REGION Network 4: Block description — Section 3.5 to 3.5
   // ▂▂▂▂▂▂▂▂▂▂▂▂▂▂▂▂▂▂▂▂▂▂▂▂▂▂▂▂▂▂▂▂▂▂▂▂▂▂▂▂▂▂▂▂
   // 3.5     Expressing the calculations in Controller operations
   // 
   // The calculations above must be rendered in a form suitable for the Simatic S7-1500 Controller, 
   // using the mathematical operations available to that Controller, these are listed in Table 2.1.
   // 
   // To perform the calculations in the Controller it will be necessary to use partial calculation to 
   // hold separate components of the overall calculation and combine these to produce the final 
   // result. 
   // 
   // The following sections breakdown each of the response calculations into these partial 
   // calculations and demonstrate how these are then combined to provide a final result that is 
   // compatible with the Controller mathematical operations and Controller notations.
   // 
   // 
   // 
   // ▁▁▁▁▁▁▁▁▁▁▁▁▁▁▁▁▁▁▁▁▁▁▁▁▁▁▁▁▁▁▁▁▁▁▁▁▁▁▁▁▁▁▁▁
   // 3.5.1     Over damped, slow response no overshoot             ζ > 1
   // 
   // 
   // CALCULATION:
   // 
   //       ╓   1 ┌   ζ       ┐   - ω [ ζ ─ √(ζ² ─ 1) ]t       1 ┌   ζ       ┐   - ω [ ζ ┼ √(ζ² ─ 1) ]t ╖
   // y(t) = K║x(t) ─ -- │------------------ ┼ 1│ｅ         ┼ -- │------------------ ─ 1│ｅ           ║
   //       ╙   2 └ √(ζ² ─ 1)     ┘            2 └ √(ζ² ─ 1)     ┘            ╜
   // 
   // 
   // 
   // Is rendered into the correct format as follows:
   // 
   // 
   //  cal_01 = SQRT ( SQR (ζ) - 1)         = √(ζ² ─ 1)
   // 
   //                                  ζ
   //  cal_02 = ζ ÷ cal_01              = -----------------
   //                          √(ζ² ─ 1)
   // 
   //  cal_03 = ζ + cal_01              = ζ ┼ √(ζ² ─ 1)
   // 
   //  cal_04 = -1 × ω × t × cal_03           = - ω [ ζ ┼ √(ζ² ─ 1) ]t
   // 
   //                              -ω [ ζ ┼ √(ζ² ─ 1) ]t 
   //  cal_05 = EXP( cal_04 )              =ｅ
   // 
   //  cal_06 = ζ - cal_01               = ζ ─ √(ζ² ─ 1)
   // 
   //  cal_07 = -1 × ω × t × cal_06           = - ω [ ζ ─ √(ζ² ─ 1) ]t
   // 
   //                            -ω [ ζ ─ √(ζ² ─ 1) ]t 
   //  cal_08 = EXP( cal_07 )              =ｅ
   // 
   //                           1 ┌   ζ       ┐
   //  cal_09 = (cal_02 - 1) × 0.5           = -- │------------------ ─ 1│
   //                           2 └ √(ζ² ─ 1)     ┘
   // 
   //                           1 ┌   ζ       ┐
   //  cal_10 = (cal_02 + 1) × 0.5            = -- │------------------ ┼ 1│
   //                           2 └ √(ζ² ─ 1)     ┘
   // 
   //                           1 ┌   ζ       ┐   -ω [ ζ ┼ √(ζ² ─ 1) ]t
   //  cal_11 = cal_09 × cal_05             = -- │------------------ ─ 1│ｅ
   //                           2 └ √(ζ² ─ 1)     ┘
   // 
   //                           1 ┌   ζ       ┐   -ω [ ζ ─ √(ζ² ─ 1) ]t
   //  cal_12 = cal_10 × cal_08             = -- │------------------ ┼ 1│ｅ
   //                           2 └ √(ζ² ─ 1)     ┘
   // 
   //                          ╓   1 ┌   ζ       ┐   - ω [ ζ ─ √(ζ² ─ 1) ]t       1 ┌   ζ       ┐   - ω [ ζ ┼ √(ζ² ─ 1) ]t ╖
   //  cal_13 = INPUT - cal_12 + cal_11        = ║x(t) ─ -- │------------------ ┼ 1│ｅ         ┼ -- │------------------ ─ 1│ｅ           ║
   //                          ╙   2 └ √(ζ² ─ 1)     ┘            2 └ √(ζ² ─ 1)     ┘            ╜
   // 
   //                             ╓   1 ┌   ζ       ┐   - ω [ ζ ─ √(ζ² ─ 1) ]t       1 ┌   ζ       ┐   - ω [ ζ ┼ √(ζ² ─ 1) ]t ╖
   //  OUTPUT  = K × cal_13             =  K║x(t) ─ -- │------------------ ┼ 1│ｅ         ┼ -- │------------------ ─ 1│ｅ           ║
   //                             ╙   2 └ √(ζ² ─ 1)     ┘            2 └ √(ζ² ─ 1)     ┘            ╜
   // 
   // 
   // 
   // ▁▁▁▁▁▁▁▁▁▁▁▁▁▁▁▁▁▁▁▁▁▁▁▁▁▁▁▁▁▁▁▁▁▁▁▁▁▁▁▁▁▁▁▁
   // 3.5.2     Critically damped, fastest response without overshoot        ζ = 1
   // 
   // 
   // CALCULATION:
   // 
   //       ╓           - ωt  ╖
   // y(t) = K║x(t) ─ (1 ┼ ωt) ｅ  ║
   //       ╙             ╜
   // 
   // 
   // Is rendered into the correct format as follows:
   // 
   // 
   //  cal_01 = -1 × ω × t                = - ωt  
   // 
   //                          - ωt
   //  cal_02 = EXP( cal_01 )              =ｅ
   // 
   //  cal_03 = 1 - cal_01              = 1 ─ (-ωt) = 1 ┼ ωt
   // 
   //                              - ωt
   //  cal_04 = cal_03 × cal_02            = (1 ┼ ωt) ｅ
   // 
   //                                 - ωt
   //  cal_05 = INPUT  - cal_04            = x(t) ─ (1 ┼ ωt) ｅ
   // 
   //                             ╓           - ωt  ╖
   //  OUTPUT  = K × cal_05             =  K║x(t) ─ (1 ┼ ωt) ｅ  ║
   //                             ╙             ╜
   // 
   // 
   // 
   // ▁▁▁▁▁▁▁▁▁▁▁▁▁▁▁▁▁▁▁▁▁▁▁▁▁▁▁▁▁▁▁▁▁▁▁▁▁▁▁▁▁▁▁▁
   // 3.5.3     Under damped, decreasing oscillations              0 < ζ < 1
   // 
   // 
   // CALCULATION:
   // 
   //       ╓      - ζω t  ┌        ζ            ┐╖
   // y(t) = K║x(t) ─ ｅ   │COS (Ωt) ┼ ------------------ SIN (Ωt)│║  where Ω =  ω √(1 ─ ζ²)
   //       ╙       └       √(1 ─ ζ²)       ┘╜
   // 
   // 
   // Is rendered into the correct format as follows:
   // 
   // 
   //  cal_01 = SQRT ( 1 - SQR (ζ))         = √(1 ─ ζ²)
   // 
   //                                  ζ
   //  cal_02 = ζ ÷ cal_01              = -----------------
   //                          √(1 ─ ζ²)
   // 
   //  cal_03 = ω × cal_01                = ω √(1 ─ ζ²) = Ω
   // 
   //  cal_04 = t × cal_03              = Ωt
   // 
   //  cal_05 = COS( cal_04 )             = COS (Ωt)
   // 
   //  cal_06 = SIN( cal_04 )               = SIN (Ωt)
   // 
   //  cal_07 = -1 × ζ × ω × t             = - ζω t 
   // 
   //                          - ζω t 
   //  cal_08 = EXP( cal_07 )              =ｅ
   // 
   //                          - ζω t 
   //  cal_09 = cal_08 × cal_05            =ｅ         COS (Ωt)
   // 
   //  
   //                                  ζ      - ζω t
   //  cal_10 = cal_02 × cal_08 × cal_06        = ----------------- ｅ         SIN (Ωt)
   //                          √(1 ─ ζ²)
   // 
   //                            ╓      - ζω t          ζ     - ζω t            ╖  ╓      - ζω t  ┌        ζ            ┐╖
   //  cal_11 = INPUT - cal_09 - cal_10          =║x(t) ─ ｅ   COS (Ωt) ─ ------------------ ｅ   SIN (Ωt)║=║x(t) ─ ｅ   │COS (Ωt) ┼ ------------------ SIN (Ωt)│║
   //                            ╙              √(1 ─ ζ²)              ╜  ╙       └       √(1 ─ ζ²)       ┘╜
   // 
   //                             ╓      - ζω t  ┌        ζ            ┐╖
   //  OUTPUT  = K × cal_11             =  K║x(t) ─ ｅ   │COS (Ωt) ┼ ------------------ SIN (Ωt)│║
   //                             ╙       └       √(1 ─ ζ²)       ┘╜
   // 
   // 
   // 
   // ▁▁▁▁▁▁▁▁▁▁▁▁▁▁▁▁▁▁▁▁▁▁▁▁▁▁▁▁▁▁▁▁▁▁▁▁▁▁▁▁▁▁▁▁
   // 3.5.4     Undamped, oscillates with frequency ω              ζ = 0
   // 
   // 
   // CALCULATION:
   // 
   //       ╓       ╖
   // y(t) = K║x(t) ─ COS (ωt) ║
   //       ╙       ╜
   // 
   // 
   // Is rendered into the correct format as follows:
   // 
   // 
   //  cal_01 = ω × t                  = ωt
   // 
   //  cal_02 = COS( cal_01 )             = COS (ωt)
   // 
   //  cal_03 = INPUT - cal_02             = x(t) ─ COS (ωt) 
   // 
   //  OUTPUT  = K × cal_03             =  K [ x(t) ─ COS (ωt) ]
   // 
   // 
   // 
   // ▁▁▁▁▁▁▁▁▁▁▁▁▁▁▁▁▁▁▁▁▁▁▁▁▁▁▁▁▁▁▁▁▁▁▁▁▁▁▁▁▁▁▁▁
   // 3.5.5     Unstable, oscillations of increasing amplitude           -1 < ζ < 0
   // 
   // 
   // CALCULATION:
   // 
   //       ╓      | ζ | ω t ┌        ζ            ┐╖
   // y(t) = K║x(t) ─ ｅ    │COS (Ωt) ┼ ------------------ SIN (Ωt)│║  where Ω =  ω √(1 ─ ζ²)
   //       ╙          └       √(1 ─ ζ²)       ┘╜
   // 
   // 
   // Is rendered into the correct format as follows:
   // 
   // 
   //  cal_01 = SQRT ( 1 - SQR (ζ))         = √(1 ─ ζ²)
   // 
   //                                  ζ
   //  cal_02 = ζ ÷ cal_01              = -----------------
   //                          √(1 ─ ζ²)
   // 
   //  cal_03 = ω × cal_01                = ω √(1 ─ ζ²) = Ω
   // 
   //  cal_04 = t × cal_03              = Ωt
   // 
   //  cal_05 = COS( cal_04 )             = COS (Ωt)
   // 
   //  cal_06 = SIN( cal_04 )               = SIN (Ωt)
   // 
   //  cal_07 = ABS(ζ) × ω × t              =  | ζ | ω t 
   // 
   //                           | ζ | ω t 
   //  cal_08 = EXP( cal_07 )              =ｅ
   // 
   //                           | ζ | ω t 
   //  cal_09 = cal_08 × cal_05            =ｅ         COS (Ωt)
   // 
   //  
   //                                  ζ      | ζ | ω t
   //  cal_10 = cal_02 × cal_08 × cal_06        = ----------------- ｅ         SIN (Ωt)
   //                          √(1 ─ ζ²)
   // 
   //                            ╓       | ζ | ω t         ζ      | ζ | ω t         ╖  ╓      | ζ | ω t ┌        ζ            ┐╖
   //  cal_11 = INPUT - cal_09 - cal_10          =║x(t) ─ ｅ   COS (Ωt) ─ ------------------ ｅ   SIN (Ωt)║=║x(t) ─ ｅ    │COS (Ωt) ┼ ------------------ SIN (Ωt)│║
   //                            ╙              √(1 ─ ζ²)              ╜  ╙        └       √(1 ─ ζ²)       ┘╜
   // 
   //                             ╓      | ζ | ω t ┌        ζ            ┐╖
   //  OUTPUT  = K × cal_11             =  K║x(t) ─ ｅ    │COS (Ωt) ┼ ------------------ SIN (Ωt)│║
   //                             ╙          └       √(1 ─ ζ²)       ┘╜
   // 
   // 
   // 
   // ▁▁▁▁▁▁▁▁▁▁▁▁▁▁▁▁▁▁▁▁▁▁▁▁▁▁▁▁▁▁▁▁▁▁▁▁▁▁▁▁▁▁▁▁
   // 3.5.6     Unstable, unbounded asymptotic increase              ζ ≤ -1
   // 
   // 
   // CALCULATION:
   // 
   //       ╓   1 ┌   ζ       ┐     ω [ | ζ | ─ √(ζ² ─ 1) ]t    1 ┌   ζ       ┐     ω [ | ζ | ┼ √(ζ² ─ 1) ]t ╖
   // y(t) = K║x(t) ─ -- │------------------ ┼ 1│ｅ         ┼ -- │------------------ ┼ 1│ｅ              ║
   //       ╙   2 └ √(ζ² ─ 1)     ┘            2 └ √(ζ² ─ 1)     ┘               ╜
   // 
   // 
   // 
   // Is rendered into the correct format as follows:
   // 
   // 
   //  cal_01 = SQRT ( SQR (ζ) - 1)         = √(ζ² ─ 1)
   // 
   //                                  ζ
   //  cal_02 = ζ ÷ cal_01              = -----------------
   //                          √(ζ² ─ 1)
   // 
   //  cal_03 = ABS (ζ) + cal_01            = | ζ | ┼ √(ζ² ─ 1)
   // 
   //  cal_04 = ω × t × cal_03             = ω [ | ζ | ┼ √(ζ² ─ 1) ]t
   // 
   //                               ω [ | ζ | ┼ √(ζ² ─ 1) ]t 
   //  cal_05 = EXP( cal_04 )              =ｅ
   // 
   //  cal_06 = ABS (ζ) - cal_01             =  | ζ | ─ √(ζ² ─ 1)
   // 
   //  cal_07 = ω × t × cal_06             = ω [  | ζ | ─ √(ζ² ─ 1) ]t
   // 
   //                               ω [  | ζ | ─ √(ζ² ─ 1) ]t 
   //  cal_08 = EXP( cal_07 )              =ｅ
   // 
   //                           1 ┌   ζ       ┐
   //  cal_09 = (cal_02 + 1) × 0.5            = -- │------------------ ┼ 1│
   //                           2 └ √(ζ² ─ 1)     ┘
   // 
   //                           1 ┌   ζ       ┐   -ω [ ζ ─ √(ζ² ─ 1) ]t
   //  cal_10 = cal_09 × cal_08             = -- │------------------ ┼ 1│ｅ
   //                           2 └ √(ζ² ─ 1)     ┘
   // 
   //                           1 ┌   ζ       ┐   -ω [ ζ ┼ √(ζ² ─ 1) ]t
   //  cal_11 = cal_09 × cal_05             = -- │------------------ ┼ 1│ｅ
   //                           2 └ √(ζ² ─ 1)     ┘
   // 
   //                          ╓   1 ┌   ζ       ┐   - ω [ ζ ─ √(ζ² ─ 1) ]t       1 ┌   ζ       ┐   - ω [ ζ ┼ √(ζ² ─ 1) ]t ╖
   //  cal_12 = INPUT - cal_10 + cal_11        = ║x(t) ─ -- │------------------ ┼ 1│ｅ         ┼ -- │------------------ ┼ 1│ｅ           ║
   //                          ╙   2 └ √(ζ² ─ 1)     ┘            2 └ √(ζ² ─ 1)     ┘            ╜
   // 
   //                             ╓   1 ┌   ζ       ┐   - ω [ ζ ─ √(ζ² ─ 1) ]t       1 ┌   ζ       ┐   - ω [ ζ ┼ √(ζ² ─ 1) ]t ╖
   //  OUTPUT  = K × cal_12             =  K║x(t) ─ -- │------------------ ┼ 1│ｅ         ┼ -- │------------------ ┼ 1│ｅ           ║
   //                             ╙   2 └ √(ζ² ─ 1)     ┘            2 └ √(ζ² ─ 1)     ┘            ╜
   // 
   // 
   // 
   // ▂▂▂▂▂▂▂▂▂▂▂▂▂▂▂▂▂▂▂▂▂▂▂▂▂▂▂▂▂▂▂▂▂▂▂▂▂▂▂▂▂▂▂▂
   // 3.6     Operating modes
   // 
   // 
   // This block FC19152_StdDebugInst2Order supports manual and automatic operating modes, the 
   // default mode is automatic.
   // 
   // The module can be switched between automatic and manual modes with the 
   // mode_AutMan signal:
   // 
   //  DATA STRUCTURE    UT39152_Dy_DebugInst2Order
   //  ――――――――――――――――――――――――――――――――――――――――――
   //  SIGNAL         FUNCTION               TYPE     DETAILS
   //  ――――――――――――――――――――――――――――――――――――――――――
   //  Mode_AutMan     Specifies the operating mode of     Bool  1 = automatic mode
   //            the simulation                 0 = manual mode
   // 
   //  Mode_Time       Specifies the manual time value of       Real     Elapsed time
   //            the simulation in seconds           in seconds
   // 
   //  status_Aut      The simulation is in automatic mode   Bool  1 = auto mode
   //                                  0 = no in auto
   // 
   //  status_Man       The simulation is in manual mode    Bool  1 = manual mode
   //                                  0 = no in manual
   //  ――――――――――――――――――――――――――――――――――――――――――  
   // 
   // 
   // 
   // ▁▁▁▁▁▁▁▁▁▁▁▁▁▁▁▁▁▁▁▁▁▁▁▁▁▁▁▁▁▁▁▁▁▁▁▁▁▁▁▁▁▁▁▁
   // 3.6.1    Automatic mode
   // 
   // 
   // By default the module will be in automatic mode. 
   // 
   // In automatic mode, if the simulation is active (TRIGGER = 1), the module carries out the relevant 
   // calculation (listed in § 3.2) depending on the value of the damping factor (k_DampFactor) each 
   // time the module is called. The module calculates the elapsed time based on the current CPU 
   // time when the module was called, compared with the CPU time when the simulation was 
   // started (rising edge of TRIGGER) and stored in actual_StartTime.
   // 
   // In automatic mode, a real time simulation occurs, generating responses similar to those shown 
   // in the plots of § 2.3.  
   // 
   // 
   // 
   // ▁▁▁▁▁▁▁▁▁▁▁▁▁▁▁▁▁▁▁▁▁▁▁▁▁▁▁▁▁▁▁▁▁▁▁▁▁▁▁▁▁▁▁▁
   // 3.6.2    Manual mode
   // 
   // 
   // In manual mode, if the simulation is active (TRIGGER = 1), the module carries out the relevant 
   // calculation (listed in § 3.2) depending on the value of the damping factor (k_DampFactor) each 
   // time the module is called; in exactly the same way as automatic mode.
   // 
   // The difference with manual mode, is that the time used in the calculation must be uniquely 
   // specified, the elapsed time is not calculated and a manual time value must be provided.
   // 
   // The manual time is given in the variable mode_ManTime and is specified in seconds.
   // 
   // If mode mode_ManTime remains constant between module calls, the module will return the 
   // same OUTPUT value each time (assuming all other signals remain unchanged).
   // 
   // Manual mode allows the module to calculate the correct response for a particular and exact time, 
   // and is not dependent on cycle times or other factors that may affect when the module is called.
   // 
   // 
   // 
   // ▁▁▁▁▁▁▁▁▁▁▁▁▁▁▁▁▁▁▁▁▁▁▁▁▁▁▁▁▁▁▁▁▁▁▁▁▁▁▁▁▁▁▁▁
   // 3.7      Symbols, block icons and faceplates
   // 
   // There is no supervisory system interface for this block. It is a debug simulation module and as
   // such has no  graphical symbol, block icon or faceplate.
   // 
   //                ━━━   ⬙⬙⬙⬙⬙⬙   ━━━
END_REGION

REGION Network 5: Block description — Sections 4 to 11
   // ▄▄▄▄▄▄▄▄▄▄▄▄▄▄▄▄▄▄▄▄▄▄▄▄▄▄▄▄▄▄▄▄▄▄▄▄▄▄▄▄▄▄▄▄
   // 4.     PARAMETERS
   // 
   // 
   // The following parameters are associated with the block:
   // 
   //  
   //  ――――――――――――――――――――――――――――――――――――――――――
   //  PARAM         FUNCTION                    TYPE      IN-OUT 
   //  ――――――――――――――――――――――――――――――――――――――――――
   //  SYS_SIGNALS      Common system signals              UT21000    In
   //           logic and timing signals for parametric access
   // 
   //  TRIGGER       Activates the simulation (the simulation will run     Bool      In
   //           whilever this signal is high), the elapsed time 
   //           is measured from the rising edge of this signal
   // 
   //  INPUT        The input time function, x(t) in the calculations     Real      In
   // 
   //  DYNAMIC_DATA      Data structure that holds the live data for the       UT39152    InOut
   //           simulation (damping factor, natural frequency, 
   //           system gain, elapsed time &c.)
   // 
   //  OUTPUT       The output time response, y(t) in the calculations   Real      Out
   //  ――――――――――――――――――――――――――――――――――――――――――
   // 
   //                ━━━   ⬙⬙⬙⬙⬙⬙   ━━━
   // 
   // 
   // 
   // ▄▄▄▄▄▄▄▄▄▄▄▄▄▄▄▄▄▄▄▄▄▄▄▄▄▄▄▄▄▄▄▄▄▄▄▄▄▄▄▄▄▄▄▄
   // 5.     DATA STRUCTURES AND USAGE (AND INSTANCE DATA BLOCKS)
   // 
   // 
   // The block has the following associated data structure:
   // 
   // 
   //  ――――――――――――――――――――――――――――――――――――――――――
   //  DATA STRUCTURE             DESCRIPTION
   //  ――――――――――――――――――――――――――――――――――――――――――
   //  UT01000_St_SysRevision          Revision information for this block    See FC01001
   //  UT01001_St_SysLicence           Licence information for this block  See FC01001
   //  UT21000_Dy_SysSignals           System signals for logic and timing  See FC01001
   // 
   //  UT39152_Dy_DebugInst2Orderl       Dynamic data storage, contains live data, such as 
   //                     calculation variables, elapsed time, oscillation 
   //                     frequency and status signals
   //  ――――――――――――――――――――――――――――――――――――――――――
   // 
   // 
   // ▂▂▂▂▂▂▂▂▂▂▂▂▂▂▂▂▂▂▂▂▂▂▂▂▂▂▂▂▂▂▂▂▂▂▂▂▂▂▂▂▂▂▂▂
   // 5.2      UT39152_Dy_DebugInst2Order
   // 
   // The static data structure for an isolating valve.
   // 
   // 
   // 
   //  UT39152_Dy_DebugInst2Order (full contents)
   //  ――――――――――――――――――――――――――――――――――――――――――
   //  SIGNAL NAME          FUNCTION                     TYPE
   //  ――――――――――――――――――――――――――――――――――――――――――
   //  k_Gain             CONSTANT — Simulation system gain        Real
   //  k_NatFreq          CONSTANT — Simulation natural frequency (rad/s)   Real
   //  k_DampFactor        CONSTANT — Simulation damping factor        Real
   //  status_Running      STATUS — Simulation is running  Bool
   //                      (1 = running, 0 = stopped)
   //  status_Stopped        STATUS — Simulation is stopped (not running)    Bool
   //                      (1 = stopped, 0 = running)
   //  status_Stable         STATUS — Simulation response type is stable     Bool
   //                      (1 = stable, 0 = unstable)
   //  status_OverDamp       STATUS — Response is stable/over damped      Bool
   //                      (1 = stable, over damped)
   //  status_CritDamp       STATUS — Response is stable/critically damped     Bool
   //                      (1 = stable, critically damped)
   //  status_UnderDamp     STATUS — Response is stable/under damped      Bool
   //                      (1 = stable, under damped)
   //  status_Undamped      STATUS — Response is stable/undamped       Bool
   //                      (1 = stable, undamped)
   //  status_USUnder        STATUS — Response is unstable/under damped    Bool
   //                      (1 = unstable, under damped)
   //  status_USOver       STATUS — Response is unstable/over damped    Bool
   //                      (1 = unstable, over damped)
   //  status_Osc          STATUS — Oscillatory response             Real
   //                      (1 = osc. response, 0 = non-osc.)
   //  status_OscFreqRS       STATUS — Frequency of oscillation, zero if       Real
   //                      non-oscillatory (rad/s)
   //  status_OscFreqHz       STATUS — Frequency of oscillation, zero if       Real
   //                      non-oscillatory (Hz)
   //  status_Period         STATUS — Period of oscillation, zero if           Real
   //                      non-oscillatory (s)
   //  status_Aut           STATUS — Simulation is in automatic mode      Bool
   //                      (1 = automatic, 0 = manual)
   //  status_Man          STATUS — Simulation is in manual mode        Bool
   //                      (1 = manual, 0 = automatic)
   //  cal_PeakValue          CALC — Peak output value             Real
   //  cal_NatPeriod        CALC — Period of natural oscillations (s)       Real
   //                    zero for non-oscillatory response
   //  cal_DampFreq       CALC — Damped frequency of the system (rad/s)    Real
   //  cal_DampFreqHz         CALC — Damped frequency of the system (Hz)     Real
   //  cal_DampPeriod       CALC — Period of damped oscillations (s)       Real
   //                    zero for non-oscillatory response
   //  cal_TimeSteady        CALC — Time to reach steady state (s)       Real
   //                    zero for unstable response
   //  cal_Time63%          CALC — Time to reach 63% of steady state (s)      Real
   //                    zero for unstable response
   //  cal_TimePeak            CALC — Time to reach the peak ouptut value (s)    Real
   //  mode_AutMan       MODE — Automatic/manual mode selection     Bool
   //                      (1 = auto mode, 0 = manual mode)
   //  mode_ManTime       MODE — Manual mode time value (s)        Real
   //  actual_StartTime         ACTUAL — CPU time when simulation started       Real
   //  actual_RunTime        ACTUAL — Elapsed time since the            Real
   //                      simulation started (s)
   //  ――――――――――――――――――――――――――――――――――――――――――
   // 
   // 
   //                ━━━   ⬙⬙⬙⬙⬙⬙   ━━━
   // 
   // 
   // 
   // ▄▄▄▄▄▄▄▄▄▄▄▄▄▄▄▄▄▄▄▄▄▄▄▄▄▄▄▄▄▄▄▄▄▄▄▄▄▄▄▄▄▄▄▄
   // 6.     CONSTANTS AND TEMPORARY (LOCAL) DATA
   // 
   // There is no constant data.
   // 
   // The following temporary data is used:
   // 
   //  Temporary (local) data
   //  ――――――――――――――――――――――――――――――――――――――――――
   //  SIGNAL NAME          FUNCTION                  TYPE
   //  ――――――――――――――――――――――――――――――――――――――――――
   //  revInfo             Revision information for the block         UT01000
   //  licInfo           Licensing information for the block      UT01001
   //  cal_01          Partial calculation see § 3.5 for details      Real
   //  cal_02          Partial calculation see § 3.5 for details      Real
   //  cal_03          Partial calculation see § 3.5 for details      Real
   //  cal_04          Partial calculation see § 3.5 for details      Real
   //  cal_05          Partial calculation see § 3.5 for details      Real
   //  cal_06          Partial calculation see § 3.5 for details      Real
   //  cal_07          Partial calculation see § 3.5 for details      Real
   //  cal_08          Partial calculation see § 3.5 for details      Real
   //  cal_09          Partial calculation see § 3.5 for details      Real
   //  cal_10          Partial calculation see § 3.5 for details      Real
   //  cal_11          Partial calculation see § 3.5 for details      Real
   //  cal_12          Partial calculation see § 3.5 for details      Real
   //  cal_13          Partial calculation see § 3.5 for details      Real
   //  wrkInt           Working storage area (integer)          Int
   //  wrkDInt           Working storage area (double integer)         DInt
   //  wrkLInt            Working storage area (long integer)        LInt
   //  wrkLTime           Working storage area (long time)         LT
   //  wrkDTL            Working storage area (DateTime long)      DTL
   //  wrkReal           Working storage (Real)             Real
   //  ―――――――――――――――――――――――――――――――――――――――――― █ █ █
   // 
   //                ━━━   ⬙⬙⬙⬙⬙⬙   ━━━
   // 
   // 
   // 
   // ▄▄▄▄▄▄▄▄▄▄▄▄▄▄▄▄▄▄▄▄▄▄▄▄▄▄▄▄▄▄▄▄▄▄▄▄▄▄▄▄▄▄▄▄
   // 7.     BLOCK CALLS
   // 
   // There are no PAL block calls from within this block.
   // 
   //                ━━━   ⬙⬙⬙⬙⬙⬙   ━━━
   // 
   // 
   // 
   // ▄▄▄▄▄▄▄▄▄▄▄▄▄▄▄▄▄▄▄▄▄▄▄▄▄▄▄▄▄▄▄▄▄▄▄▄▄▄▄▄▄▄▄▄
   // 8.     ASSOCIATED BLOCKS
   // 
   // 
   // This is a stand-alone block and is not associated with any other blocks.
   // 
   //                ━━━   ⬙⬙⬙⬙⬙⬙   ━━━
   // 
   // 
   // 
   // ▄▄▄▄▄▄▄▄▄▄▄▄▄▄▄▄▄▄▄▄▄▄▄▄▄▄▄▄▄▄▄▄▄▄▄▄▄▄▄▄▄▄▄▄
   // 9.     SYSTEM BLOCK CALLS AND SYSTEM DATA TYPES
   // 
   // The following calls are made to system blocks:
   // 
   // 
   //  System block calls
   //  ――――――――――――――――――――――――――――――――――――――――――
   //  BLOCK          TITLE             DESCRIPTION  
   //  ――――――――――――――――――――――――――――――――――――――――――
   //  RD_LOC_T             Read the local RTC time    Reads the CPU real time clock 
   //  ――――――――――――――――――――――――――――――――――――――――――
   // 
   // There are no special system data types used.
   // 
   // 
   //                ━━━   ⬙⬙⬙⬙⬙⬙   ━━━
   // 
   // 
   // 
   // ▄▄▄▄▄▄▄▄▄▄▄▄▄▄▄▄▄▄▄▄▄▄▄▄▄▄▄▄▄▄▄▄▄▄▄▄▄▄▄▄▄▄▄▄
   // 10.     SPECIAL PROPERTIES AND REQUIREMENTS
   // 
   // 
   // 
   // ▂▂▂▂▂▂▂▂▂▂▂▂▂▂▂▂▂▂▂▂▂▂▂▂▂▂▂▂▂▂▂▂▂▂▂▂▂▂▂▂▂▂▂▂
   // 10.1   Block optimisation
   // 
   // 
   // Block optimisation is ACTIVE for this block
   // 
   // 
   // 
   // ▂▂▂▂▂▂▂▂▂▂▂▂▂▂▂▂▂▂▂▂▂▂▂▂▂▂▂▂▂▂▂▂▂▂▂▂▂▂▂▂▂▂▂▂
   // 10.2   Calling requirements
   // 
   // 
   // There are no special calling requirements for this block.
   // 
   //                ━━━   ⬙⬙⬙⬙⬙⬙   ━━━
   // 
   // 
   // 
   // ▄▄▄▄▄▄▄▄▄▄▄▄▄▄▄▄▄▄▄▄▄▄▄▄▄▄▄▄▄▄▄▄▄▄▄▄▄▄▄▄▄▄▄▄
   // 11.     EXAMPLE USAGE
   // 
   // 
   // The following shows a typical deployment of FC19512:
   // 
   //                         ┌─────────────
   //      ───────────────────┤ FC19512
   //                         ├───────────────┤
   //    "DB21001_DY_StdGlobalData".SysSignals ─┤ SYS_SIGNALS            
   //                         │               OUTPUT ├─  "wrk_Real"
   //                         │               │
   //                                                        "1.0" ─┤ INPUT                     │
   //                         │               │
   //                   %M999.0     │               │
   //                    "SIM01_TRIG" ─┤ TRIGGER                     │
   //                         │               │
   //                         │
   //       "DB39152_Dy_DebugInst2Order".S001 ─┤ DYNAMIC_DATA
   //                         │
   //                         │
   //                                         │
   //                                ─────────┘
   // 
   // 
   //               ━━━   ⬙⬙⬙⬙⬙⬙   ━━━
   // 
   // 
   // ██████████████ █ █ █ █  END   █ █ █ █ ██████████████
END_REGION

REGION Network 6: Current revision and modification history
   // ▄▄▄▄▄▄▄▄▄▄▄▄▄▄▄▄▄▄▄▄▄▄▄▄▄▄▄▄▄▄▄▄▄▄▄▄▄▄▄▄▄▄▄▄
   // MODIFICATION HISTORY
   // 
   // 
   // The revision data shown here, in the network comments, contains additional information 
   // reflecting the software development workflow under the version control system (VCS) employed 
   // to track all software changes.
   // 
   // The VCS in use is the Git Source Code Management system in conjunction with the GitHub online 
   // hosting system. The software in its entirety is available in the GitHub remote repository:
   // 
   //      https://github.com/practicalseries/PS2001-pal-software
   // 
   // The repository is public and can be freely copied (forked in GitHub terminology) and used 
   // under the MIT licence. 
   // 
   // The MIT licence is reproduced in full in the last network of this software module.
   // 
   // 
   //  ―――――――――――――――――――――――――――――――――――――――――――
   //  DATE       REVISION             MASTER BRANCH     DEV
   //          (nnn.amm)   COMMIT TAG    (Base ---> Merge)    BRANCH   Author
   //  ———————————————————————————————————————————
   //  2022.01.12    000.101   D0009A-000.101   D0009 N/A     D0009A   M. Gledhill
   //                        FC19512 Block created — Comments added
   //  ———————————————————————————————————————————
   //   Where: nnn  =  Major revision
   //         a  =  Type (1-7 Development, 8 Proving, 9 Qualification, 0 Release)
   //       mm  =  Minor revision (must be 00 if a = 0)
   //         Block properties version number should be set to nn.a (only one decimal place)
   // 
   // ▄▄▄▄▄▄▄▄▄▄▄▄▄▄▄▄▄▄▄▄▄▄▄▄▄▄▄▄▄▄▄▄▄▄▄▄▄▄▄▄▄▄▄▄
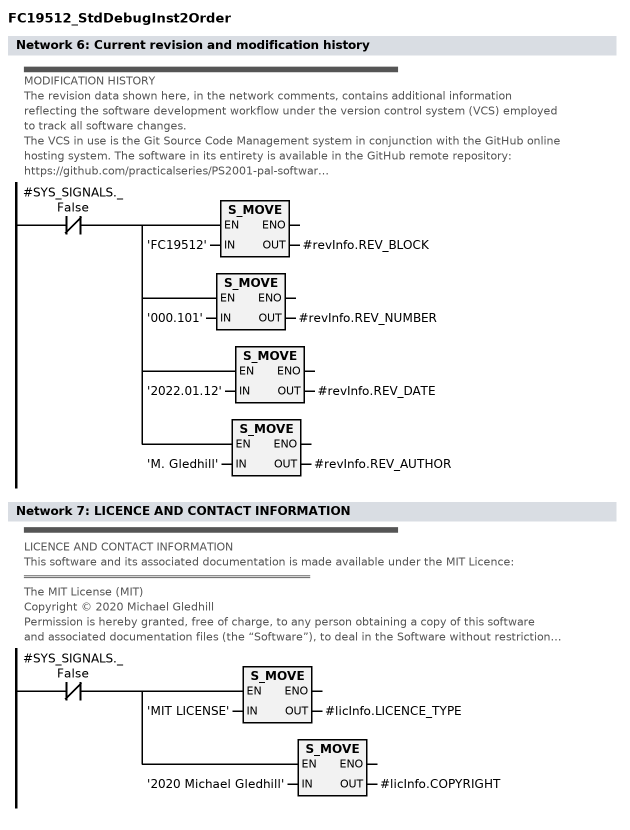
   RUNG wire#powerrail
      I_Contact( #SYS_SIGNALS._False )
      wire#w1
      S_Move(in := 'FC19512', out => #revInfo.REV_BLOCK)
   END_RUNG
   RUNG wire#w1
      S_Move(in := '000.101', out => #revInfo.REV_NUMBER)
   END_RUNG
   RUNG wire#w1
      S_Move(in := '2022.01.12', out => #revInfo.REV_DATE)
   END_RUNG
   RUNG wire#w1
      S_Move(in := 'M. Gledhill', out => #revInfo.REV_AUTHOR)
   END_RUNG
   // the same network as SCL:
   IF NOT #SYS_SIGNALS._False THEN
       #revInfo.REV_BLOCK := 'FC19512';
       #revInfo.REV_NUMBER := '000.101';
       #revInfo.REV_DATE := '2022.01.12';
       #revInfo.REV_AUTHOR := 'M. Gledhill';
   END_IF;
END_REGION

REGION Network 7: LICENCE AND CONTACT INFORMATION
   // ▀▀▀▀▀▀▀▀▀▀▀▀▀▀▀▀▀▀▀▀▀▀▀▀▀▀▀▀▀▀▀▀▀▀▀▀▀▀▀▀▀▀▀▀
   // LICENCE AND CONTACT INFORMATION
   // 
   // This software and its associated documentation is made available under the MIT Licence:
   // 
   // ════════════════════════════════════════════
   // 
   // The MIT License (MIT)
   // 
   // Copyright © 2020 Michael Gledhill
   // 
   // Permission is hereby granted, free of charge, to any person obtaining a copy of this software 
   // and associated documentation files (the “Software”), to deal in the Software without restriction, 
   // including without limitation the rights to use, copy, modify, merge, publish, distribute, 
   // sublicense, and/or sell copies of the Software, and to permit persons to whom the Software is 
   // furnished to do so, subject to the following conditions: 
   // 
   // The above copyright notice and this permission notice shall be included in all copies or 
   // substantial portions of the Software.
   // 
   // THE SOFTWARE IS PROVIDED “AS IS”, WITHOUT WARRANTY OF ANY KIND, EXPRESS OR IMPLIED, 
   // INCLUDING BUT NOT LIMITED TO THE WARRANTIES OF MERCHANTABILITY, FITNESS FOR A 
   // PARTICULAR PURPOSE AND NON-INFRINGEMENT. IN NO EVENT SHALL THE AUTHORS OR COPYRIGHT 
   // HOLDERS BE LIABLE FOR ANY CLAIM, DAMAGES OR OTHER LIABILITY, WHETHER IN AN ACTION OF 
   // CONTRACT, TORT OR OTHERWISE, ARISING FROM, OUT OF OR IN CONNECTION WITH THE SOFTWARE 
   // OR THE USE OR OTHER DEALINGS IN THE SOFTWARE.
   // 
   // ════════════════════════════════════════════
   //                    ┌────────────┐
   // You can reach the author by email here:   │  mg@practicalseries.com  │
   //                    └────────────┘
   // Questions, corrections, constructive criticism and complaints (polite ones) are invited.
   RUNG wire#powerrail
      I_Contact( #SYS_SIGNALS._False )
      wire#w1
      S_Move(in := 'MIT LICENSE', out => #licInfo.LICENCE_TYPE)
   END_RUNG
   RUNG wire#w1
      S_Move(in := '2020 Michael Gledhill', out => #licInfo.COPYRIGHT)
   END_RUNG
   // the same network as SCL:
   IF NOT #SYS_SIGNALS._False THEN
       #licInfo.LICENCE_TYPE := 'MIT LICENSE';
       #licInfo.COPYRIGHT := '2020 Michael Gledhill';
   END_IF;
END_REGION
END_FUNCTION
